TYPE ST125_PnpHorPos_e : ST120_PnpHorPos_e;
END_TYPE

(* stored: Version 1.1.0.1, ProductVersion 3.1.4024.6
   DUT ST125_PnpHorPos_e: Id {bf1edbb1-6055-4f77-94f4-33abebdf517b} *)
